ABB RAPID module: Wobj_rfl_locexp_mdfplate3.mod

MODULE Wobj_rfl_locexp_mdfplate3
	! Points are read in order of declaration.
  ! Please do not change the order of points!

  LOCAL PERS robtarget pWobj_U_PointX1:=[[1677.642,-286.2471,-523.6169],[0.205883786082268,0.583549499511719,0.774832367897034,0.129292860627174],[-1,-3,2,0],[9E+09,9E+09,9E+09,9E+09,9E+09,9E+09]];
	LOCAL PERS robtarget pWobj_U_PointX2:=[[1700.495,-896.7616,-520.1512],[0.204200774431229,0.577883541584015,0.773908793926239,0.159429550170898],[-1,-3,-1,0],[9E+09,9E+09,9E+09,9E+09,9E+09,9E+09]];
	LOCAL PERS robtarget pWobj_U_PointY1:=[[1682.396,-283.5428,565.8287],[0.480135649442673,0.543206453323364,0.640085399150848,0.254336655139923],[-1,0,0,1],[9E+09,9E+09,9E+09,9E+09,9E+09,9E+09]];

ENDMODULE
